# EPICS substitutions: gemBeamlineJawsApp/Db/gem_beamline_jawset.substitutions
global {P=\$(P), MOD_TO_SAMPLE=\$(MOD_TO_SAMPLE)}

file "$(TOP)/jawsManagerApp/Db/common.template" {
	{DIR=H}
	{DIR=V}
}

file "$(TOP)/jawsManagerApp/Db/jaws_manager_single.template" {
    {JAW="JAWS1", MOD_TO_JAW="\$(MOD_TO_JAWS1)"}
    {JAW="JAWS2", MOD_TO_JAW="\$(MOD_TO_JAWS2)"}
    {JAW="JAWS3", MOD_TO_JAW="\$(MOD_TO_JAWS3)"}
    {JAW="JAWS4", MOD_TO_JAW="\$(MOD_TO_JAWS4)"}
	{JAW="JAWS5", MOD_TO_JAW="\$(MOD_TO_JAWS5)"}
}
